FUNCTION_BLOCK Stage6 (* Template for a Basic Function Block Type *)
  (* Standard: 61499-2 *)
  (* Version 1.0, 2021-06-20, HP *)
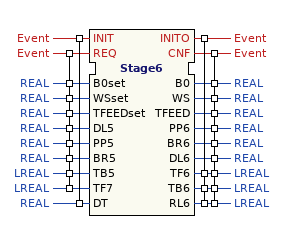
  EVENT_INPUT
    INIT WITH DT; (* Initialization Request *)
    REQ WITH B0set, WSset, TFEEDset, DL5, PP5, BR5, TB5, TF7; (* Normal Execution Request *)
  END_EVENT
  EVENT_OUTPUT
    INITO WITH TB6, RL6, TF6; (* Initialization Confirm *)
    CNF WITH TB6, DL6, TF6, BR6, PP6, B0, WS, TFEED, RL6; (* Execution Confirmation *)
  END_EVENT
  VAR_INPUT
    B0set : REAL;
    WSset : REAL;
    TFEEDset : REAL;
    DL5 : REAL;
    PP5 : REAL;
    BR5 : REAL;
    TB5 : LREAL;
    TF7 : LREAL;
    DT : REAL;
  END_VAR
  VAR_OUTPUT
    B0 : REAL;
    WS : REAL;
    TFEED : REAL;
    PP6 : REAL;
    BR6 : REAL;
    DL6 : REAL;
    TF6 : LREAL;
    TB6 : LREAL;
    RL6 : LREAL;
  END_VAR
  VAR
    AB : REAL; (* internal variabel *)
    UU : REAL;
    TREF : REAL;
    AD : REAL;
    AHC : REAL;
    AHR : REAL;
    AS : REAL;
    REC : REAL;
    WN : REAL;
    WN_1 : REAL;
    XKN : REAL;
    C1 : REAL;
    HS : REAL;
    G : REAL;
    W1 : REAL;
    TFREC : REAL;
    TS : REAL;
    DTS : REAL;
    TF6_last : REAL;
    RL6_last : REAL;
    TB6_last : REAL;
    USS : REAL;
    RHOB : REAL;
    CPB : REAL;
    CPF : REAL;
    FMW : REAL;
    HLV : REAL;
    HV : REAL;
    BPR : REAL;
    FMC : REAL;
    U : REAL;
    A : REAL;
    B : REAL;
    C : REAL;
    D1 : REAL;
    d : REAL;
    a : REAL;
    A1 : REAL;
    A2 : REAL;
    A3 : REAL;
    A4 : REAL;
    A5 : REAL;
    A6 : REAL;
    p : REAL;
    q : REAL;
    TC : REAL;
    PC : REAL;
    DTB6 : REAL;
    DEN6 : REAL;
    DH6 : REAL;
    DP6 : REAL;
    DPDH6 : REAL;
    DT6 : REAL;
    m : REAL;
    n : REAL;
    VR6 : REAL;
    DELTA6 : REAL;
    DELTA28 : REAL;
    DELTA50 : REAL;
    DELTA6_last : REAL;
    DELTA28_last : REAL;
    DELTA50_last : REAL;
  END_VAR
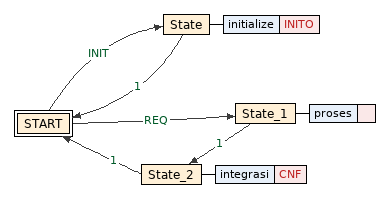
  EC_STATES
    START; (* Initial State *)
    State : initialize -> INITO;
    State_1 : proses;
    State_2 : integrasi -> CNF;
  END_STATES
  EC_TRANSITIONS
    START TO State := INIT;
    State TO START := 1;
    START TO State_1 := REQ;
    State_1 TO State_2 := 1;
    State_2 TO START := 1;
  END_TRANSITIONS
  ALGORITHM initialize IN ST: (* Initialization algorithm *)
TREF :=273.15;
AB :=57.2727;
AHC :=4069.2;
AHR :=2639.7;
AS :=3225.7;
REC :=0.0;
//TF2:=TF2;

//TFEED :=TFEED1+TREF;
 //TS:=TS1+TREF;
WN :=3.0;
XKN :=0.68;
HS:=0.11;
G :=9.81;
W1 :=0.50;

RL6 := 0.545579116884776;
TB6 := 351.066232011349;
TF6 := 347.148389575489;
TF7 := 344.515318586845;


RL6_last :=RL6;
TB6_last :=TB6;
TF6_last :=TF6;
  END_ALGORITHM
  ALGORITHM proses IN ST: (* kalkulasi *)
B0 :=B0set;
WS :=WSset;
TFEED:=TFEEDset;
UU := TFEEDset;
U :=UU;

USS :=49.767;
C1 :=0.625;
RHOB :=1032.4; //maassa jenis brine
CPB :=1.00; //heatcapacity Brine
CPF :=1.00; //heat capacity feed
FMW :=23654.0;
HLV :=563.7959;
HV :=625.1971;
BPR :=2.192;
FMC :=34736.09;
//U :=UU; //feed temp



///  Calculate the physical properties

//A :=3.2437814;
//B :=5.86826*0.001;
//C :=1.1702379*0.00000001;
//D1 :=2.1878462*0.001;
//TC :=647.27;
//PC :=218.167;


A1 :=3.2437814;
A2:=5.86826*0.001;
A3:=1.1702379*0.00000001;
A4 :=2.1878462*0.001;
A5 :=647.27;
A6 :=218.167;

DTB6 :=A5-TB6;
DEN6 :=(A1+A2*DTB6+A3*DTB6*DTB6*DTB6)/(1+A4*DTB6)*DTB6/TB6;
p:=DEN6;
q:=10.0;
PP6 :=A6/(EXPT(q, p));

// calculate the brine flow rates
DP6:=PP5-PP6;
DH6:=RL6-C1*HS;
DPDH6 :=DP6*101000+G*RHOB*DH6;
m:=DPDH6*RHOB;
n:=0.5;
BR6 :=WN*XKN*RL6*(EXPT(m, n));
BR6 :=BR6*60.0/1000.0;

// calculate the vapor flow rates

DT6 :=TB6-BPR/1.8-(TF7+TF6)*0.5;
VR6 :=U*AHC*DT6/HLV/1000.0;
DL6 :=DL5+VR6;


//// state equation
DELTA6 :=(BR5-BR6-VR6)*1000.0/RHOB/AB;
DELTA28 :=((BR5*CPB*(TB5-TB6))-VR6*(HV-CPB*(TB6-TREF)))*1000.0/AB/RHOB/CPB/RL6;
DELTA50 :=(B0*CPF*(TF7-TF6)*1000+(U*AHC*DT6))/FMW/CPF;
  END_ALGORITHM
  ALGORITHM integrasi IN ST: (* new algorithm *)
B0 :=B0set;
WS :=WSset;
TFEED:=TFEEDset;
//integrasi
RL6 := (DELTA6 + DELTA6_last)*0.5*DT + RL6_last;
DELTA6_last :=DELTA6 ;
RL6_last :=RL6;

TB6 := (DELTA28 + DELTA28_last)*0.5*DT + TB6_last;
DELTA28_last :=DELTA28 ;
TB6_last:=TB6;

TF6 := (DELTA50 + DELTA50_last)*0.5*DT + TF6_last;
DELTA50_last :=DELTA50 ;
TF6_last :=TF6;
  END_ALGORITHM
END_FUNCTION_BLOCK
